(* IEC 61131-3 sources: codesys4-agent-guide/examples/minimal/Minimal.fbsdev/Application.iecapp^, 1 file *)

(* ---- PLC_PRG.prg.st ---- *)
// Minimal example: counts PLC cycles. Same shape as the UI's PLC_PRG template.
PROGRAM PLC_PRG
VAR
    nCycles : UDINT;
END_VAR

nCycles := nCycles + 1;

END_PROGRAM
